// TIA Portal V19 export
FUNCTION "FC40_CommSlave" : Void   // FC40, LAD
{ S7_Optimized_Access := 'TRUE' }
// stored: AutoNumber false, IsIECCheckEnabled true, SetENOAutomatically false
BEGIN

REGION Network 1: Manage communication with Left PLC
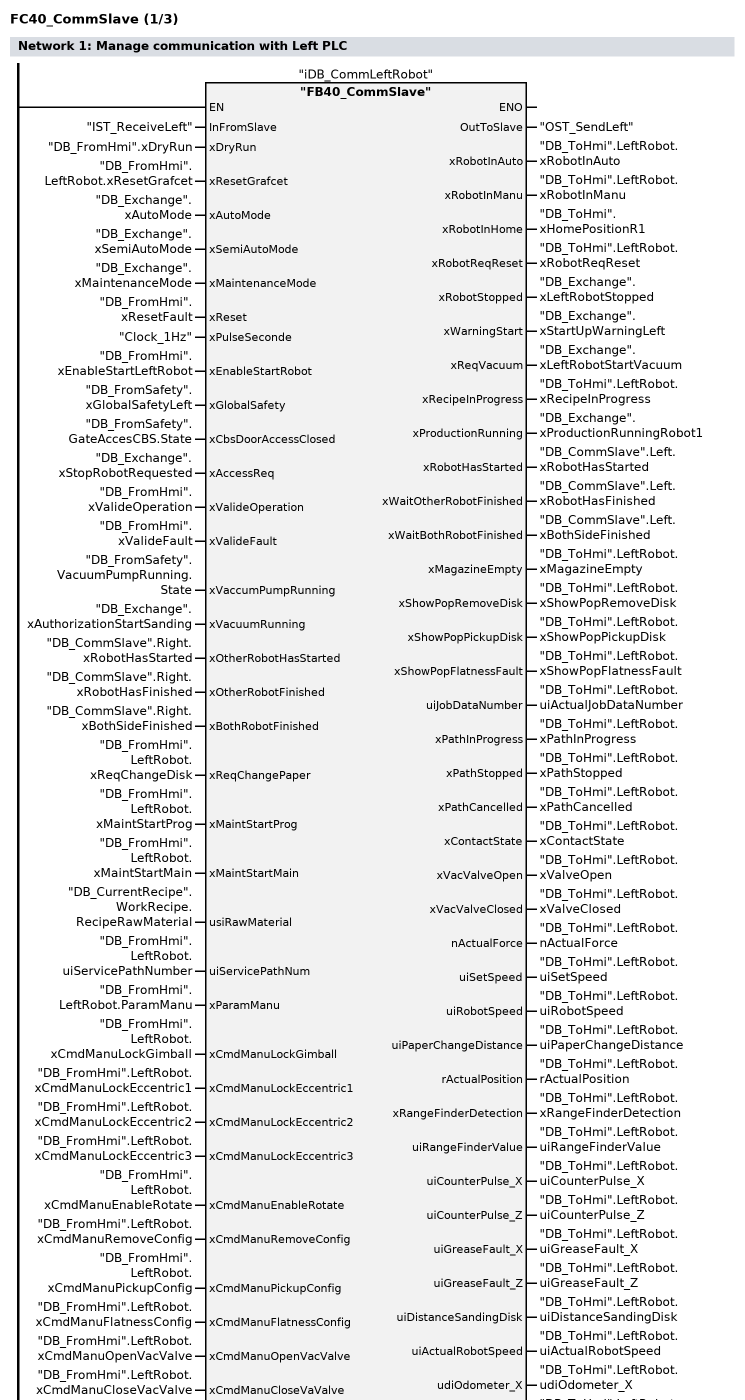
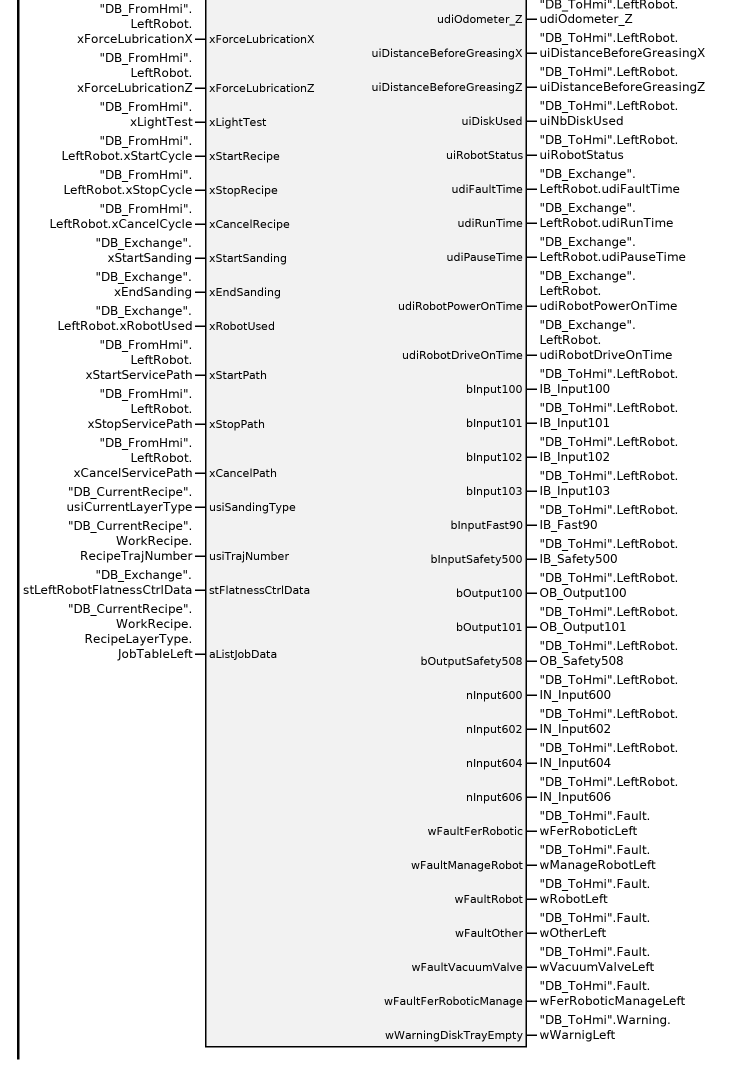
   RUNG wire#powerrail
      "iDB_CommLeftRobot"(InFromSlave := "IST_ReceiveLeft", xDryRun := "DB_FromHmi".xDryRun, xResetGrafcet := "DB_FromHmi".LeftRobot.xResetGrafcet, xAutoMode := "DB_Exchange".xAutoMode, xSemiAutoMode := "DB_Exchange".xSemiAutoMode, xMaintenanceMode := "DB_Exchange".xMaintenanceMode, xReset := "DB_FromHmi".xResetFault, xPulseSeconde := "Clock_1Hz", xEnableStartRobot := "DB_FromHmi".xEnableStartLeftRobot, xGlobalSafety := "DB_FromSafety".xGlobalSafetyLeft, xCbsDoorAccessClosed := "DB_FromSafety".GateAccesCBS.State, xAccessReq := "DB_Exchange".xStopRobotRequested, xValideOperation := "DB_FromHmi".xValideOperation, xValideFault := "DB_FromHmi".xValideFault, xVaccumPumpRunning := "DB_FromSafety".VacuumPumpRunning.State, xVacuumRunning := "DB_Exchange".xAuthorizationStartSanding, xOtherRobotHasStarted := "DB_CommSlave".Right.xRobotHasStarted, xOtherRobotFinished := "DB_CommSlave".Right.xRobotHasFinished, xBothRobotFinished := "DB_CommSlave".Right.xBothSideFinished, xReqChangePaper := "DB_FromHmi".LeftRobot.xReqChangeDisk, xMaintStartProg := "DB_FromHmi".LeftRobot.xMaintStartProg, xMaintStartMain := "DB_FromHmi".LeftRobot.xMaintStartMain, usiRawMaterial := "DB_CurrentRecipe".WorkRecipe.RecipeRawMaterial, uiServicePathNum := "DB_FromHmi".LeftRobot.uiServicePathNumber, xParamManu := "DB_FromHmi".LeftRobot.ParamManu, xCmdManuLockGimball := "DB_FromHmi".LeftRobot.xCmdManuLockGimball, xCmdManuLockEccentric1 := "DB_FromHmi".LeftRobot.xCmdManuLockEccentric1, xCmdManuLockEccentric2 := "DB_FromHmi".LeftRobot.xCmdManuLockEccentric2, xCmdManuLockEccentric3 := "DB_FromHmi".LeftRobot.xCmdManuLockEccentric3, xCmdManuEnableRotate := "DB_FromHmi".LeftRobot.xCmdManuEnableRotate, xCmdManuRemoveConfig := "DB_FromHmi".LeftRobot.xCmdManuRemoveConfig, xCmdManuPickupConfig := "DB_FromHmi".LeftRobot.xCmdManuPickupConfig, xCmdManuFlatnessConfig := "DB_FromHmi".LeftRobot.xCmdManuFlatnessConfig, xCmdManuOpenVacValve := "DB_FromHmi".LeftRobot.xCmdManuOpenVacValve, xCmdManuCloseVaValve := "DB_FromHmi".LeftRobot.xCmdManuCloseVacValve, xForceLubricationX := "DB_FromHmi".LeftRobot.xForceLubricationX, xForceLubricationZ := "DB_FromHmi".LeftRobot.xForceLubricationZ, xLightTest := "DB_FromHmi".xLightTest, xStartRecipe := "DB_FromHmi".LeftRobot.xStartCycle, xStopRecipe := "DB_FromHmi".LeftRobot.xStopCycle, xCancelRecipe := "DB_FromHmi".LeftRobot.xCancelCycle, xStartSanding := "DB_Exchange".xStartSanding, xEndSanding := "DB_Exchange".xEndSanding, xRobotUsed := "DB_Exchange".LeftRobot.xRobotUsed, xStartPath := "DB_FromHmi".LeftRobot.xStartServicePath, xStopPath := "DB_FromHmi".LeftRobot.xStopServicePath, xCancelPath := "DB_FromHmi".LeftRobot.xCancelServicePath, usiSandingType := "DB_CurrentRecipe".usiCurrentLayerType, usiTrajNumber := "DB_CurrentRecipe".WorkRecipe.RecipeTrajNumber, stFlatnessCtrlData := "DB_Exchange".stLeftRobotFlatnessCtrlData, aListJobData := "DB_CurrentRecipe".WorkRecipe.RecipeLayerType.JobTableLeft, OutToSlave => "OST_SendLeft", xRobotInAuto => "DB_ToHmi".LeftRobot.xRobotInAuto, xRobotInManu => "DB_ToHmi".LeftRobot.xRobotInManu, xRobotInHome => "DB_ToHmi".xHomePositionR1, xRobotReqReset => "DB_ToHmi".LeftRobot.xRobotReqReset, xRobotStopped => "DB_Exchange".xLeftRobotStopped, xWarningStart => "DB_Exchange".xStartUpWarningLeft, xReqVacuum => "DB_Exchange".xLeftRobotStartVacuum, xRecipeInProgress => "DB_ToHmi".LeftRobot.xRecipeInProgress, xProductionRunning => "DB_Exchange".xProductionRunningRobot1, xRobotHasStarted => "DB_CommSlave".Left.xRobotHasStarted, xWaitOtherRobotFinished => "DB_CommSlave".Left.xRobotHasFinished, xWaitBothRobotFinished => "DB_CommSlave".Left.xBothSideFinished, xMagazineEmpty => "DB_ToHmi".LeftRobot.xMagazineEmpty, xShowPopRemoveDisk => "DB_ToHmi".LeftRobot.xShowPopRemoveDisk, xShowPopPickupDisk => "DB_ToHmi".LeftRobot.xShowPopPickupDisk, xShowPopFlatnessFault => "DB_ToHmi".LeftRobot.xShowPopFlatnessFault, uiJobDataNumber => "DB_ToHmi".LeftRobot.uiActualJobDataNumber, xPathInProgress => "DB_ToHmi".LeftRobot.xPathInProgress, xPathStopped => "DB_ToHmi".LeftRobot.xPathStopped, xPathCancelled => "DB_ToHmi".LeftRobot.xPathCancelled, xContactState => "DB_ToHmi".LeftRobot.xContactState, xVacValveOpen => "DB_ToHmi".LeftRobot.xValveOpen, xVacValveClosed => "DB_ToHmi".LeftRobot.xValveClosed, nActualForce => "DB_ToHmi".LeftRobot.nActualForce, uiSetSpeed => "DB_ToHmi".LeftRobot.uiSetSpeed, uiRobotSpeed => "DB_ToHmi".LeftRobot.uiRobotSpeed, uiPaperChangeDistance => "DB_ToHmi".LeftRobot.uiPaperChangeDistance, rActualPosition => "DB_ToHmi".LeftRobot.rActualPosition, xRangeFinderDetection => "DB_ToHmi".LeftRobot.xRangeFinderDetection, uiRangeFinderValue => "DB_ToHmi".LeftRobot.uiRangeFinderValue, uiCounterPulse_X => "DB_ToHmi".LeftRobot.uiCounterPulse_X, uiCounterPulse_Z => "DB_ToHmi".LeftRobot.uiCounterPulse_Z, uiGreaseFault_X => "DB_ToHmi".LeftRobot.uiGreaseFault_X, uiGreaseFault_Z => "DB_ToHmi".LeftRobot.uiGreaseFault_Z, uiDistanceSandingDisk => "DB_ToHmi".LeftRobot.uiDistanceSandingDisk, uiActualRobotSpeed => "DB_ToHmi".LeftRobot.uiActualRobotSpeed, udiOdometer_X => "DB_ToHmi".LeftRobot.udiOdometer_X, udiOdometer_Z => "DB_ToHmi".LeftRobot.udiOdometer_Z, uiDistanceBeforeGreasingX => "DB_ToHmi".LeftRobot.uiDistanceBeforeGreasingX, uiDistanceBeforeGreasingZ => "DB_ToHmi".LeftRobot.uiDistanceBeforeGreasingZ, uiDiskUsed => "DB_ToHmi".LeftRobot.uiNbDiskUsed, uiRobotStatus => "DB_ToHmi".LeftRobot.uiRobotStatus, udiFaultTime => "DB_Exchange".LeftRobot.udiFaultTime, udiRunTime => "DB_Exchange".LeftRobot.udiRunTime, udiPauseTime => "DB_Exchange".LeftRobot.udiPauseTime, udiRobotPowerOnTime => "DB_Exchange".LeftRobot.udiRobotPowerOnTime, udiRobotDriveOnTime => "DB_Exchange".LeftRobot.udiRobotDriveOnTime, bInput100 => "DB_ToHmi".LeftRobot.IB_Input100, bInput101 => "DB_ToHmi".LeftRobot.IB_Input101, bInput102 => "DB_ToHmi".LeftRobot.IB_Input102, bInput103 => "DB_ToHmi".LeftRobot.IB_Input103, bInputFast90 => "DB_ToHmi".LeftRobot.IB_Fast90, bInputSafety500 => "DB_ToHmi".LeftRobot.IB_Safety500, bOutput100 => "DB_ToHmi".LeftRobot.OB_Output100, bOutput101 => "DB_ToHmi".LeftRobot.OB_Output101, bOutputSafety508 => "DB_ToHmi".LeftRobot.OB_Safety508, nInput600 => "DB_ToHmi".LeftRobot.IN_Input600, nInput602 => "DB_ToHmi".LeftRobot.IN_Input602, nInput604 => "DB_ToHmi".LeftRobot.IN_Input604, nInput606 => "DB_ToHmi".LeftRobot.IN_Input606, wFaultFerRobotic => "DB_ToHmi".Fault.wFerRoboticLeft, wFaultManageRobot => "DB_ToHmi".Fault.wManageRobotLeft, wFaultRobot => "DB_ToHmi".Fault.wRobotLeft, wFaultOther => "DB_ToHmi".Fault.wOtherLeft, wFaultVacuumValve => "DB_ToHmi".Fault.wVacuumValveLeft, wFaultFerRoboticManage => "DB_ToHmi".Fault.wFerRoboticManageLeft, wWarningDiskTrayEmpty => "DB_ToHmi".Warning.wWarnigLeft)
   END_RUNG
   // the same network as SCL:
   "iDB_CommLeftRobot"(InFromSlave := "IST_ReceiveLeft",   // "FB40_CommSlave"
                       xDryRun := "DB_FromHmi".xDryRun,
                       xResetGrafcet := "DB_FromHmi".LeftRobot.xResetGrafcet,
                       xAutoMode := "DB_Exchange".xAutoMode,
                       xSemiAutoMode := "DB_Exchange".xSemiAutoMode,
                       xMaintenanceMode := "DB_Exchange".xMaintenanceMode,
                       xReset := "DB_FromHmi".xResetFault,
                       xPulseSeconde := "Clock_1Hz",
                       xEnableStartRobot := "DB_FromHmi".xEnableStartLeftRobot,
                       xGlobalSafety := "DB_FromSafety".xGlobalSafetyLeft,
                       xCbsDoorAccessClosed := "DB_FromSafety".GateAccesCBS.State,
                       xAccessReq := "DB_Exchange".xStopRobotRequested,
                       xValideOperation := "DB_FromHmi".xValideOperation,
                       xValideFault := "DB_FromHmi".xValideFault,
                       xVaccumPumpRunning := "DB_FromSafety".VacuumPumpRunning.State,
                       xVacuumRunning := "DB_Exchange".xAuthorizationStartSanding,
                       xOtherRobotHasStarted := "DB_CommSlave".Right.xRobotHasStarted,
                       xOtherRobotFinished := "DB_CommSlave".Right.xRobotHasFinished,
                       xBothRobotFinished := "DB_CommSlave".Right.xBothSideFinished,
                       xReqChangePaper := "DB_FromHmi".LeftRobot.xReqChangeDisk,
                       xMaintStartProg := "DB_FromHmi".LeftRobot.xMaintStartProg,
                       xMaintStartMain := "DB_FromHmi".LeftRobot.xMaintStartMain,
                       usiRawMaterial := "DB_CurrentRecipe".WorkRecipe.RecipeRawMaterial,
                       uiServicePathNum := "DB_FromHmi".LeftRobot.uiServicePathNumber,
                       xParamManu := "DB_FromHmi".LeftRobot.ParamManu,
                       xCmdManuLockGimball := "DB_FromHmi".LeftRobot.xCmdManuLockGimball,
                       xCmdManuLockEccentric1 := "DB_FromHmi".LeftRobot.xCmdManuLockEccentric1,
                       xCmdManuLockEccentric2 := "DB_FromHmi".LeftRobot.xCmdManuLockEccentric2,
                       xCmdManuLockEccentric3 := "DB_FromHmi".LeftRobot.xCmdManuLockEccentric3,
                       xCmdManuEnableRotate := "DB_FromHmi".LeftRobot.xCmdManuEnableRotate,
                       xCmdManuRemoveConfig := "DB_FromHmi".LeftRobot.xCmdManuRemoveConfig,
                       xCmdManuPickupConfig := "DB_FromHmi".LeftRobot.xCmdManuPickupConfig,
                       xCmdManuFlatnessConfig := "DB_FromHmi".LeftRobot.xCmdManuFlatnessConfig,
                       xCmdManuOpenVacValve := "DB_FromHmi".LeftRobot.xCmdManuOpenVacValve,
                       xCmdManuCloseVaValve := "DB_FromHmi".LeftRobot.xCmdManuCloseVacValve,
                       xForceLubricationX := "DB_FromHmi".LeftRobot.xForceLubricationX,
                       xForceLubricationZ := "DB_FromHmi".LeftRobot.xForceLubricationZ,
                       xLightTest := "DB_FromHmi".xLightTest,
                       xStartRecipe := "DB_FromHmi".LeftRobot.xStartCycle,
                       xStopRecipe := "DB_FromHmi".LeftRobot.xStopCycle,
                       xCancelRecipe := "DB_FromHmi".LeftRobot.xCancelCycle,
                       xStartSanding := "DB_Exchange".xStartSanding,
                       xEndSanding := "DB_Exchange".xEndSanding,
                       xRobotUsed := "DB_Exchange".LeftRobot.xRobotUsed,
                       xStartPath := "DB_FromHmi".LeftRobot.xStartServicePath,
                       xStopPath := "DB_FromHmi".LeftRobot.xStopServicePath,
                       xCancelPath := "DB_FromHmi".LeftRobot.xCancelServicePath,
                       usiSandingType := "DB_CurrentRecipe".usiCurrentLayerType,
                       usiTrajNumber := "DB_CurrentRecipe".WorkRecipe.RecipeTrajNumber,
                       stFlatnessCtrlData := "DB_Exchange".stLeftRobotFlatnessCtrlData,
                       aListJobData := "DB_CurrentRecipe".WorkRecipe.RecipeLayerType.JobTableLeft,
                       OutToSlave => "OST_SendLeft",
                       xRobotInAuto => "DB_ToHmi".LeftRobot.xRobotInAuto,
                       xRobotInManu => "DB_ToHmi".LeftRobot.xRobotInManu,
                       xRobotInHome => "DB_ToHmi".xHomePositionR1,
                       xRobotReqReset => "DB_ToHmi".LeftRobot.xRobotReqReset,
                       xRobotStopped => "DB_Exchange".xLeftRobotStopped,
                       xWarningStart => "DB_Exchange".xStartUpWarningLeft,
                       xReqVacuum => "DB_Exchange".xLeftRobotStartVacuum,
                       xRecipeInProgress => "DB_ToHmi".LeftRobot.xRecipeInProgress,
                       xProductionRunning => "DB_Exchange".xProductionRunningRobot1,
                       xRobotHasStarted => "DB_CommSlave".Left.xRobotHasStarted,
                       xWaitOtherRobotFinished => "DB_CommSlave".Left.xRobotHasFinished,
                       xWaitBothRobotFinished => "DB_CommSlave".Left.xBothSideFinished,
                       xMagazineEmpty => "DB_ToHmi".LeftRobot.xMagazineEmpty,
                       xShowPopRemoveDisk => "DB_ToHmi".LeftRobot.xShowPopRemoveDisk,
                       xShowPopPickupDisk => "DB_ToHmi".LeftRobot.xShowPopPickupDisk,
                       xShowPopFlatnessFault => "DB_ToHmi".LeftRobot.xShowPopFlatnessFault,
                       uiJobDataNumber => "DB_ToHmi".LeftRobot.uiActualJobDataNumber,
                       xPathInProgress => "DB_ToHmi".LeftRobot.xPathInProgress,
                       xPathStopped => "DB_ToHmi".LeftRobot.xPathStopped,
                       xPathCancelled => "DB_ToHmi".LeftRobot.xPathCancelled,
                       xContactState => "DB_ToHmi".LeftRobot.xContactState,
                       xVacValveOpen => "DB_ToHmi".LeftRobot.xValveOpen,
                       xVacValveClosed => "DB_ToHmi".LeftRobot.xValveClosed,
                       nActualForce => "DB_ToHmi".LeftRobot.nActualForce,
                       uiSetSpeed => "DB_ToHmi".LeftRobot.uiSetSpeed,
                       uiRobotSpeed => "DB_ToHmi".LeftRobot.uiRobotSpeed,
                       uiPaperChangeDistance => "DB_ToHmi".LeftRobot.uiPaperChangeDistance,
                       rActualPosition => "DB_ToHmi".LeftRobot.rActualPosition,
                       xRangeFinderDetection => "DB_ToHmi".LeftRobot.xRangeFinderDetection,
                       uiRangeFinderValue => "DB_ToHmi".LeftRobot.uiRangeFinderValue,
                       uiCounterPulse_X => "DB_ToHmi".LeftRobot.uiCounterPulse_X,
                       uiCounterPulse_Z => "DB_ToHmi".LeftRobot.uiCounterPulse_Z,
                       uiGreaseFault_X => "DB_ToHmi".LeftRobot.uiGreaseFault_X,
                       uiGreaseFault_Z => "DB_ToHmi".LeftRobot.uiGreaseFault_Z,
                       uiDistanceSandingDisk => "DB_ToHmi".LeftRobot.uiDistanceSandingDisk,
                       uiActualRobotSpeed => "DB_ToHmi".LeftRobot.uiActualRobotSpeed,
                       udiOdometer_X => "DB_ToHmi".LeftRobot.udiOdometer_X,
                       udiOdometer_Z => "DB_ToHmi".LeftRobot.udiOdometer_Z,
                       uiDistanceBeforeGreasingX => "DB_ToHmi".LeftRobot.uiDistanceBeforeGreasingX,
                       uiDistanceBeforeGreasingZ => "DB_ToHmi".LeftRobot.uiDistanceBeforeGreasingZ,
                       uiDiskUsed => "DB_ToHmi".LeftRobot.uiNbDiskUsed,
                       uiRobotStatus => "DB_ToHmi".LeftRobot.uiRobotStatus,
                       udiFaultTime => "DB_Exchange".LeftRobot.udiFaultTime,
                       udiRunTime => "DB_Exchange".LeftRobot.udiRunTime,
                       udiPauseTime => "DB_Exchange".LeftRobot.udiPauseTime,
                       udiRobotPowerOnTime => "DB_Exchange".LeftRobot.udiRobotPowerOnTime,
                       udiRobotDriveOnTime => "DB_Exchange".LeftRobot.udiRobotDriveOnTime,
                       bInput100 => "DB_ToHmi".LeftRobot.IB_Input100,
                       bInput101 => "DB_ToHmi".LeftRobot.IB_Input101,
                       bInput102 => "DB_ToHmi".LeftRobot.IB_Input102,
                       bInput103 => "DB_ToHmi".LeftRobot.IB_Input103,
                       bInputFast90 => "DB_ToHmi".LeftRobot.IB_Fast90,
                       bInputSafety500 => "DB_ToHmi".LeftRobot.IB_Safety500,
                       bOutput100 => "DB_ToHmi".LeftRobot.OB_Output100,
                       bOutput101 => "DB_ToHmi".LeftRobot.OB_Output101,
                       bOutputSafety508 => "DB_ToHmi".LeftRobot.OB_Safety508,
                       nInput600 => "DB_ToHmi".LeftRobot.IN_Input600,
                       nInput602 => "DB_ToHmi".LeftRobot.IN_Input602,
                       nInput604 => "DB_ToHmi".LeftRobot.IN_Input604,
                       nInput606 => "DB_ToHmi".LeftRobot.IN_Input606,
                       wFaultFerRobotic => "DB_ToHmi".Fault.wFerRoboticLeft,
                       wFaultManageRobot => "DB_ToHmi".Fault.wManageRobotLeft,
                       wFaultRobot => "DB_ToHmi".Fault.wRobotLeft,
                       wFaultOther => "DB_ToHmi".Fault.wOtherLeft,
                       wFaultVacuumValve => "DB_ToHmi".Fault.wVacuumValveLeft,
                       wFaultFerRoboticManage => "DB_ToHmi".Fault.wFerRoboticManageLeft,
                       wWarningDiskTrayEmpty => "DB_ToHmi".Warning.wWarnigLeft);
END_REGION

REGION Network 2: Manage communication with Right PLC
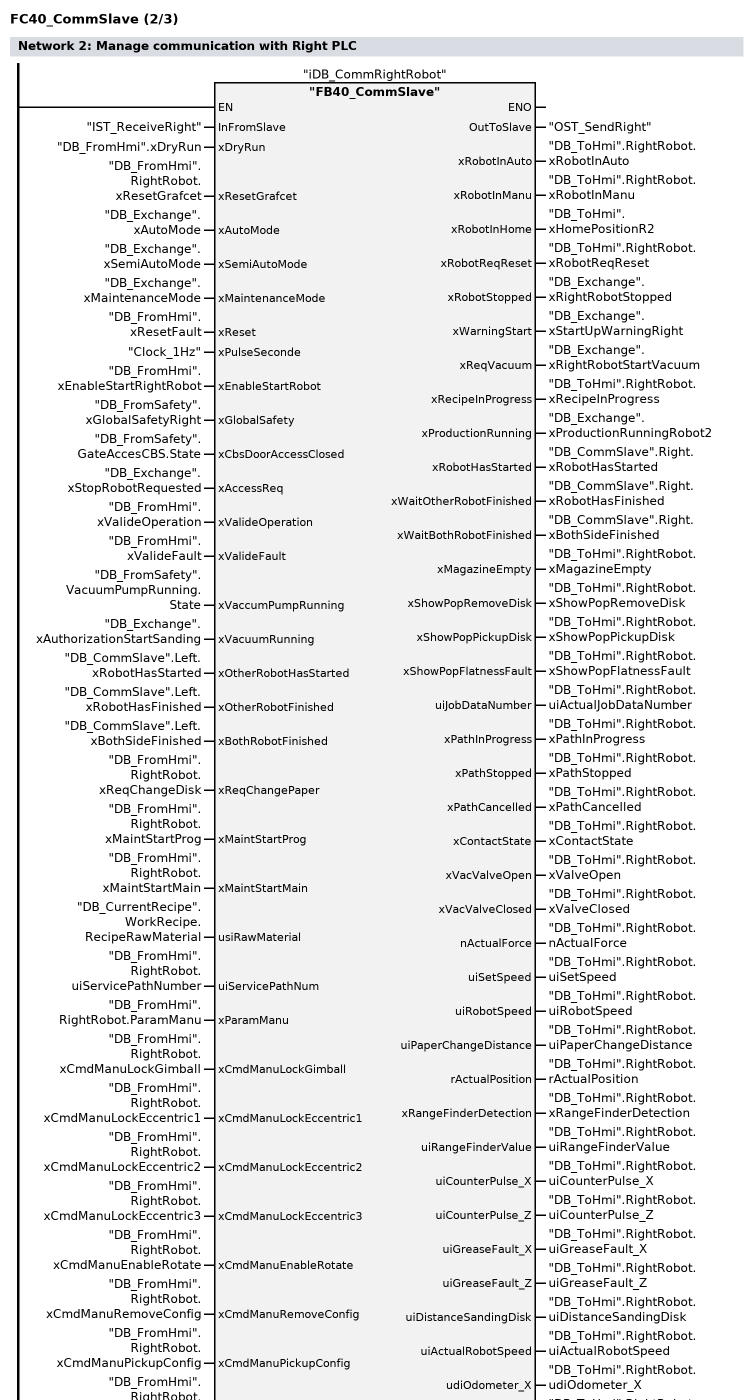
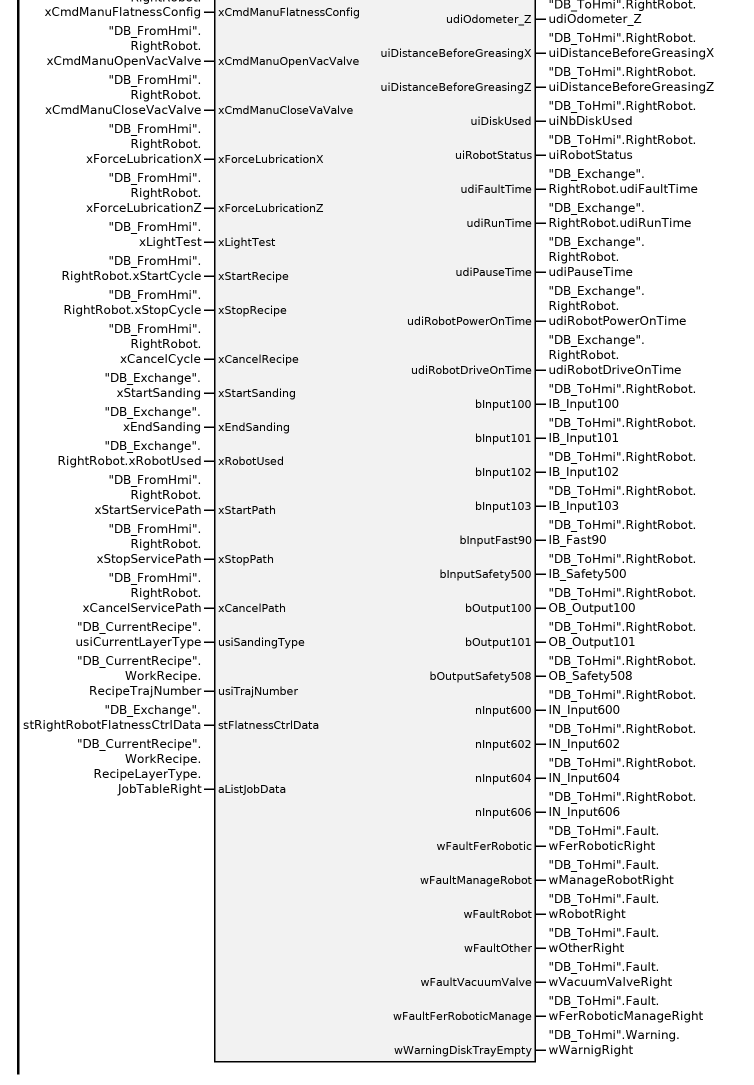
   RUNG wire#powerrail
      "iDB_CommRightRobot"(InFromSlave := "IST_ReceiveRight", xDryRun := "DB_FromHmi".xDryRun, xResetGrafcet := "DB_FromHmi".RightRobot.xResetGrafcet, xAutoMode := "DB_Exchange".xAutoMode, xSemiAutoMode := "DB_Exchange".xSemiAutoMode, xMaintenanceMode := "DB_Exchange".xMaintenanceMode, xReset := "DB_FromHmi".xResetFault, xPulseSeconde := "Clock_1Hz", xEnableStartRobot := "DB_FromHmi".xEnableStartRightRobot, xGlobalSafety := "DB_FromSafety".xGlobalSafetyRight, xCbsDoorAccessClosed := "DB_FromSafety".GateAccesCBS.State, xAccessReq := "DB_Exchange".xStopRobotRequested, xValideOperation := "DB_FromHmi".xValideOperation, xValideFault := "DB_FromHmi".xValideFault, xVaccumPumpRunning := "DB_FromSafety".VacuumPumpRunning.State, xVacuumRunning := "DB_Exchange".xAuthorizationStartSanding, xOtherRobotHasStarted := "DB_CommSlave".Left.xRobotHasStarted, xOtherRobotFinished := "DB_CommSlave".Left.xRobotHasFinished, xBothRobotFinished := "DB_CommSlave".Left.xBothSideFinished, xReqChangePaper := "DB_FromHmi".RightRobot.xReqChangeDisk, xMaintStartProg := "DB_FromHmi".RightRobot.xMaintStartProg, xMaintStartMain := "DB_FromHmi".RightRobot.xMaintStartMain, usiRawMaterial := "DB_CurrentRecipe".WorkRecipe.RecipeRawMaterial, uiServicePathNum := "DB_FromHmi".RightRobot.uiServicePathNumber, xParamManu := "DB_FromHmi".RightRobot.ParamManu, xCmdManuLockGimball := "DB_FromHmi".RightRobot.xCmdManuLockGimball, xCmdManuLockEccentric1 := "DB_FromHmi".RightRobot.xCmdManuLockEccentric1, xCmdManuLockEccentric2 := "DB_FromHmi".RightRobot.xCmdManuLockEccentric2, xCmdManuLockEccentric3 := "DB_FromHmi".RightRobot.xCmdManuLockEccentric3, xCmdManuEnableRotate := "DB_FromHmi".RightRobot.xCmdManuEnableRotate, xCmdManuRemoveConfig := "DB_FromHmi".RightRobot.xCmdManuRemoveConfig, xCmdManuPickupConfig := "DB_FromHmi".RightRobot.xCmdManuPickupConfig, xCmdManuFlatnessConfig := "DB_FromHmi".RightRobot.xCmdManuFlatnessConfig, xCmdManuOpenVacValve := "DB_FromHmi".RightRobot.xCmdManuOpenVacValve, xCmdManuCloseVaValve := "DB_FromHmi".RightRobot.xCmdManuCloseVacValve, xForceLubricationX := "DB_FromHmi".RightRobot.xForceLubricationX, xForceLubricationZ := "DB_FromHmi".RightRobot.xForceLubricationZ, xLightTest := "DB_FromHmi".xLightTest, xStartRecipe := "DB_FromHmi".RightRobot.xStartCycle, xStopRecipe := "DB_FromHmi".RightRobot.xStopCycle, xCancelRecipe := "DB_FromHmi".RightRobot.xCancelCycle, xStartSanding := "DB_Exchange".xStartSanding, xEndSanding := "DB_Exchange".xEndSanding, xRobotUsed := "DB_Exchange".RightRobot.xRobotUsed, xStartPath := "DB_FromHmi".RightRobot.xStartServicePath, xStopPath := "DB_FromHmi".RightRobot.xStopServicePath, xCancelPath := "DB_FromHmi".RightRobot.xCancelServicePath, usiSandingType := "DB_CurrentRecipe".usiCurrentLayerType, usiTrajNumber := "DB_CurrentRecipe".WorkRecipe.RecipeTrajNumber, stFlatnessCtrlData := "DB_Exchange".stRightRobotFlatnessCtrlData, aListJobData := "DB_CurrentRecipe".WorkRecipe.RecipeLayerType.JobTableRight, OutToSlave => "OST_SendRight", xRobotInAuto => "DB_ToHmi".RightRobot.xRobotInAuto, xRobotInManu => "DB_ToHmi".RightRobot.xRobotInManu, xRobotInHome => "DB_ToHmi".xHomePositionR2, xRobotReqReset => "DB_ToHmi".RightRobot.xRobotReqReset, xRobotStopped => "DB_Exchange".xRightRobotStopped, xWarningStart => "DB_Exchange".xStartUpWarningRight, xReqVacuum => "DB_Exchange".xRightRobotStartVacuum, xRecipeInProgress => "DB_ToHmi".RightRobot.xRecipeInProgress, xProductionRunning => "DB_Exchange".xProductionRunningRobot2, xRobotHasStarted => "DB_CommSlave".Right.xRobotHasStarted, xWaitOtherRobotFinished => "DB_CommSlave".Right.xRobotHasFinished, xWaitBothRobotFinished => "DB_CommSlave".Right.xBothSideFinished, xMagazineEmpty => "DB_ToHmi".RightRobot.xMagazineEmpty, xShowPopRemoveDisk => "DB_ToHmi".RightRobot.xShowPopRemoveDisk, xShowPopPickupDisk => "DB_ToHmi".RightRobot.xShowPopPickupDisk, xShowPopFlatnessFault => "DB_ToHmi".RightRobot.xShowPopFlatnessFault, uiJobDataNumber => "DB_ToHmi".RightRobot.uiActualJobDataNumber, xPathInProgress => "DB_ToHmi".RightRobot.xPathInProgress, xPathStopped => "DB_ToHmi".RightRobot.xPathStopped, xPathCancelled => "DB_ToHmi".RightRobot.xPathCancelled, xContactState => "DB_ToHmi".RightRobot.xContactState, xVacValveOpen => "DB_ToHmi".RightRobot.xValveOpen, xVacValveClosed => "DB_ToHmi".RightRobot.xValveClosed, nActualForce => "DB_ToHmi".RightRobot.nActualForce, uiSetSpeed => "DB_ToHmi".RightRobot.uiSetSpeed, uiRobotSpeed => "DB_ToHmi".RightRobot.uiRobotSpeed, uiPaperChangeDistance => "DB_ToHmi".RightRobot.uiPaperChangeDistance, rActualPosition => "DB_ToHmi".RightRobot.rActualPosition, xRangeFinderDetection => "DB_ToHmi".RightRobot.xRangeFinderDetection, uiRangeFinderValue => "DB_ToHmi".RightRobot.uiRangeFinderValue, uiCounterPulse_X => "DB_ToHmi".RightRobot.uiCounterPulse_X, uiCounterPulse_Z => "DB_ToHmi".RightRobot.uiCounterPulse_Z, uiGreaseFault_X => "DB_ToHmi".RightRobot.uiGreaseFault_X, uiGreaseFault_Z => "DB_ToHmi".RightRobot.uiGreaseFault_Z, uiDistanceSandingDisk => "DB_ToHmi".RightRobot.uiDistanceSandingDisk, uiActualRobotSpeed => "DB_ToHmi".RightRobot.uiActualRobotSpeed, udiOdometer_X => "DB_ToHmi".RightRobot.udiOdometer_X, udiOdometer_Z => "DB_ToHmi".RightRobot.udiOdometer_Z, uiDistanceBeforeGreasingX => "DB_ToHmi".RightRobot.uiDistanceBeforeGreasingX, uiDistanceBeforeGreasingZ => "DB_ToHmi".RightRobot.uiDistanceBeforeGreasingZ, uiDiskUsed => "DB_ToHmi".RightRobot.uiNbDiskUsed, uiRobotStatus => "DB_ToHmi".RightRobot.uiRobotStatus, udiFaultTime => "DB_Exchange".RightRobot.udiFaultTime, udiRunTime => "DB_Exchange".RightRobot.udiRunTime, udiPauseTime => "DB_Exchange".RightRobot.udiPauseTime, udiRobotPowerOnTime => "DB_Exchange".RightRobot.udiRobotPowerOnTime, udiRobotDriveOnTime => "DB_Exchange".RightRobot.udiRobotDriveOnTime, bInput100 => "DB_ToHmi".RightRobot.IB_Input100, bInput101 => "DB_ToHmi".RightRobot.IB_Input101, bInput102 => "DB_ToHmi".RightRobot.IB_Input102, bInput103 => "DB_ToHmi".RightRobot.IB_Input103, bInputFast90 => "DB_ToHmi".RightRobot.IB_Fast90, bInputSafety500 => "DB_ToHmi".RightRobot.IB_Safety500, bOutput100 => "DB_ToHmi".RightRobot.OB_Output100, bOutput101 => "DB_ToHmi".RightRobot.OB_Output101, bOutputSafety508 => "DB_ToHmi".RightRobot.OB_Safety508, nInput600 => "DB_ToHmi".RightRobot.IN_Input600, nInput602 => "DB_ToHmi".RightRobot.IN_Input602, nInput604 => "DB_ToHmi".RightRobot.IN_Input604, nInput606 => "DB_ToHmi".RightRobot.IN_Input606, wFaultFerRobotic => "DB_ToHmi".Fault.wFerRoboticRight, wFaultManageRobot => "DB_ToHmi".Fault.wManageRobotRight, wFaultRobot => "DB_ToHmi".Fault.wRobotRight, wFaultOther => "DB_ToHmi".Fault.wOtherRight, wFaultVacuumValve => "DB_ToHmi".Fault.wVacuumValveRight, wFaultFerRoboticManage => "DB_ToHmi".Fault.wFerRoboticManageRight, wWarningDiskTrayEmpty => "DB_ToHmi".Warning.wWarnigRight)
   END_RUNG
   // the same network as SCL:
   "iDB_CommRightRobot"(InFromSlave := "IST_ReceiveRight",   // "FB40_CommSlave"
                        xDryRun := "DB_FromHmi".xDryRun,
                        xResetGrafcet := "DB_FromHmi".RightRobot.xResetGrafcet,
                        xAutoMode := "DB_Exchange".xAutoMode,
                        xSemiAutoMode := "DB_Exchange".xSemiAutoMode,
                        xMaintenanceMode := "DB_Exchange".xMaintenanceMode,
                        xReset := "DB_FromHmi".xResetFault,
                        xPulseSeconde := "Clock_1Hz",
                        xEnableStartRobot := "DB_FromHmi".xEnableStartRightRobot,
                        xGlobalSafety := "DB_FromSafety".xGlobalSafetyRight,
                        xCbsDoorAccessClosed := "DB_FromSafety".GateAccesCBS.State,
                        xAccessReq := "DB_Exchange".xStopRobotRequested,
                        xValideOperation := "DB_FromHmi".xValideOperation,
                        xValideFault := "DB_FromHmi".xValideFault,
                        xVaccumPumpRunning := "DB_FromSafety".VacuumPumpRunning.State,
                        xVacuumRunning := "DB_Exchange".xAuthorizationStartSanding,
                        xOtherRobotHasStarted := "DB_CommSlave".Left.xRobotHasStarted,
                        xOtherRobotFinished := "DB_CommSlave".Left.xRobotHasFinished,
                        xBothRobotFinished := "DB_CommSlave".Left.xBothSideFinished,
                        xReqChangePaper := "DB_FromHmi".RightRobot.xReqChangeDisk,
                        xMaintStartProg := "DB_FromHmi".RightRobot.xMaintStartProg,
                        xMaintStartMain := "DB_FromHmi".RightRobot.xMaintStartMain,
                        usiRawMaterial := "DB_CurrentRecipe".WorkRecipe.RecipeRawMaterial,
                        uiServicePathNum := "DB_FromHmi".RightRobot.uiServicePathNumber,
                        xParamManu := "DB_FromHmi".RightRobot.ParamManu,
                        xCmdManuLockGimball := "DB_FromHmi".RightRobot.xCmdManuLockGimball,
                        xCmdManuLockEccentric1 := "DB_FromHmi".RightRobot.xCmdManuLockEccentric1,
                        xCmdManuLockEccentric2 := "DB_FromHmi".RightRobot.xCmdManuLockEccentric2,
                        xCmdManuLockEccentric3 := "DB_FromHmi".RightRobot.xCmdManuLockEccentric3,
                        xCmdManuEnableRotate := "DB_FromHmi".RightRobot.xCmdManuEnableRotate,
                        xCmdManuRemoveConfig := "DB_FromHmi".RightRobot.xCmdManuRemoveConfig,
                        xCmdManuPickupConfig := "DB_FromHmi".RightRobot.xCmdManuPickupConfig,
                        xCmdManuFlatnessConfig := "DB_FromHmi".RightRobot.xCmdManuFlatnessConfig,
                        xCmdManuOpenVacValve := "DB_FromHmi".RightRobot.xCmdManuOpenVacValve,
                        xCmdManuCloseVaValve := "DB_FromHmi".RightRobot.xCmdManuCloseVacValve,
                        xForceLubricationX := "DB_FromHmi".RightRobot.xForceLubricationX,
                        xForceLubricationZ := "DB_FromHmi".RightRobot.xForceLubricationZ,
                        xLightTest := "DB_FromHmi".xLightTest,
                        xStartRecipe := "DB_FromHmi".RightRobot.xStartCycle,
                        xStopRecipe := "DB_FromHmi".RightRobot.xStopCycle,
                        xCancelRecipe := "DB_FromHmi".RightRobot.xCancelCycle,
                        xStartSanding := "DB_Exchange".xStartSanding,
                        xEndSanding := "DB_Exchange".xEndSanding,
                        xRobotUsed := "DB_Exchange".RightRobot.xRobotUsed,
                        xStartPath := "DB_FromHmi".RightRobot.xStartServicePath,
                        xStopPath := "DB_FromHmi".RightRobot.xStopServicePath,
                        xCancelPath := "DB_FromHmi".RightRobot.xCancelServicePath,
                        usiSandingType := "DB_CurrentRecipe".usiCurrentLayerType,
                        usiTrajNumber := "DB_CurrentRecipe".WorkRecipe.RecipeTrajNumber,
                        stFlatnessCtrlData := "DB_Exchange".stRightRobotFlatnessCtrlData,
                        aListJobData := "DB_CurrentRecipe".WorkRecipe.RecipeLayerType.JobTableRight,
                        OutToSlave => "OST_SendRight",
                        xRobotInAuto => "DB_ToHmi".RightRobot.xRobotInAuto,
                        xRobotInManu => "DB_ToHmi".RightRobot.xRobotInManu,
                        xRobotInHome => "DB_ToHmi".xHomePositionR2,
                        xRobotReqReset => "DB_ToHmi".RightRobot.xRobotReqReset,
                        xRobotStopped => "DB_Exchange".xRightRobotStopped,
                        xWarningStart => "DB_Exchange".xStartUpWarningRight,
                        xReqVacuum => "DB_Exchange".xRightRobotStartVacuum,
                        xRecipeInProgress => "DB_ToHmi".RightRobot.xRecipeInProgress,
                        xProductionRunning => "DB_Exchange".xProductionRunningRobot2,
                        xRobotHasStarted => "DB_CommSlave".Right.xRobotHasStarted,
                        xWaitOtherRobotFinished => "DB_CommSlave".Right.xRobotHasFinished,
                        xWaitBothRobotFinished => "DB_CommSlave".Right.xBothSideFinished,
                        xMagazineEmpty => "DB_ToHmi".RightRobot.xMagazineEmpty,
                        xShowPopRemoveDisk => "DB_ToHmi".RightRobot.xShowPopRemoveDisk,
                        xShowPopPickupDisk => "DB_ToHmi".RightRobot.xShowPopPickupDisk,
                        xShowPopFlatnessFault => "DB_ToHmi".RightRobot.xShowPopFlatnessFault,
                        uiJobDataNumber => "DB_ToHmi".RightRobot.uiActualJobDataNumber,
                        xPathInProgress => "DB_ToHmi".RightRobot.xPathInProgress,
                        xPathStopped => "DB_ToHmi".RightRobot.xPathStopped,
                        xPathCancelled => "DB_ToHmi".RightRobot.xPathCancelled,
                        xContactState => "DB_ToHmi".RightRobot.xContactState,
                        xVacValveOpen => "DB_ToHmi".RightRobot.xValveOpen,
                        xVacValveClosed => "DB_ToHmi".RightRobot.xValveClosed,
                        nActualForce => "DB_ToHmi".RightRobot.nActualForce,
                        uiSetSpeed => "DB_ToHmi".RightRobot.uiSetSpeed,
                        uiRobotSpeed => "DB_ToHmi".RightRobot.uiRobotSpeed,
                        uiPaperChangeDistance => "DB_ToHmi".RightRobot.uiPaperChangeDistance,
                        rActualPosition => "DB_ToHmi".RightRobot.rActualPosition,
                        xRangeFinderDetection => "DB_ToHmi".RightRobot.xRangeFinderDetection,
                        uiRangeFinderValue => "DB_ToHmi".RightRobot.uiRangeFinderValue,
                        uiCounterPulse_X => "DB_ToHmi".RightRobot.uiCounterPulse_X,
                        uiCounterPulse_Z => "DB_ToHmi".RightRobot.uiCounterPulse_Z,
                        uiGreaseFault_X => "DB_ToHmi".RightRobot.uiGreaseFault_X,
                        uiGreaseFault_Z => "DB_ToHmi".RightRobot.uiGreaseFault_Z,
                        uiDistanceSandingDisk => "DB_ToHmi".RightRobot.uiDistanceSandingDisk,
                        uiActualRobotSpeed => "DB_ToHmi".RightRobot.uiActualRobotSpeed,
                        udiOdometer_X => "DB_ToHmi".RightRobot.udiOdometer_X,
                        udiOdometer_Z => "DB_ToHmi".RightRobot.udiOdometer_Z,
                        uiDistanceBeforeGreasingX => "DB_ToHmi".RightRobot.uiDistanceBeforeGreasingX,
                        uiDistanceBeforeGreasingZ => "DB_ToHmi".RightRobot.uiDistanceBeforeGreasingZ,
                        uiDiskUsed => "DB_ToHmi".RightRobot.uiNbDiskUsed,
                        uiRobotStatus => "DB_ToHmi".RightRobot.uiRobotStatus,
                        udiFaultTime => "DB_Exchange".RightRobot.udiFaultTime,
                        udiRunTime => "DB_Exchange".RightRobot.udiRunTime,
                        udiPauseTime => "DB_Exchange".RightRobot.udiPauseTime,
                        udiRobotPowerOnTime => "DB_Exchange".RightRobot.udiRobotPowerOnTime,
                        udiRobotDriveOnTime => "DB_Exchange".RightRobot.udiRobotDriveOnTime,
                        bInput100 => "DB_ToHmi".RightRobot.IB_Input100,
                        bInput101 => "DB_ToHmi".RightRobot.IB_Input101,
                        bInput102 => "DB_ToHmi".RightRobot.IB_Input102,
                        bInput103 => "DB_ToHmi".RightRobot.IB_Input103,
                        bInputFast90 => "DB_ToHmi".RightRobot.IB_Fast90,
                        bInputSafety500 => "DB_ToHmi".RightRobot.IB_Safety500,
                        bOutput100 => "DB_ToHmi".RightRobot.OB_Output100,
                        bOutput101 => "DB_ToHmi".RightRobot.OB_Output101,
                        bOutputSafety508 => "DB_ToHmi".RightRobot.OB_Safety508,
                        nInput600 => "DB_ToHmi".RightRobot.IN_Input600,
                        nInput602 => "DB_ToHmi".RightRobot.IN_Input602,
                        nInput604 => "DB_ToHmi".RightRobot.IN_Input604,
                        nInput606 => "DB_ToHmi".RightRobot.IN_Input606,
                        wFaultFerRobotic => "DB_ToHmi".Fault.wFerRoboticRight,
                        wFaultManageRobot => "DB_ToHmi".Fault.wManageRobotRight,
                        wFaultRobot => "DB_ToHmi".Fault.wRobotRight,
                        wFaultOther => "DB_ToHmi".Fault.wOtherRight,
                        wFaultVacuumValve => "DB_ToHmi".Fault.wVacuumValveRight,
                        wFaultFerRoboticManage => "DB_ToHmi".Fault.wFerRoboticManageRight,
                        wWarningDiskTrayEmpty => "DB_ToHmi".Warning.wWarnigRight);
END_REGION

REGION Network 3: Sanding process is in progress
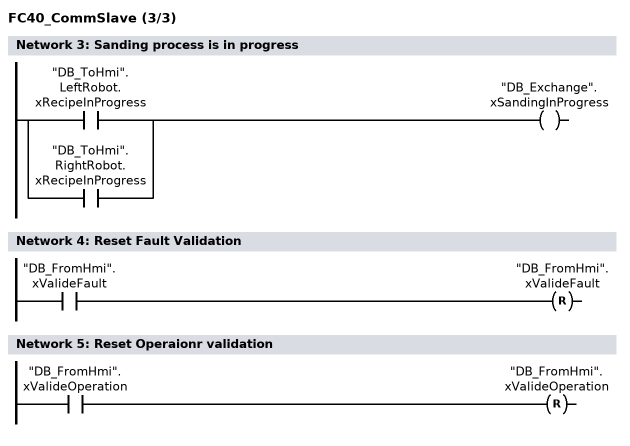
   RUNG wire#powerrail
      Contact( "DB_ToHmi".LeftRobot.xRecipeInProgress )
      wire#w1
      Coil( "DB_Exchange".xSandingInProgress )
   END_RUNG
   RUNG wire#powerrail
      Contact( "DB_ToHmi".RightRobot.xRecipeInProgress )
   END_RUNG wire#w1
   // the same network as SCL:
   "DB_Exchange".xSandingInProgress := "DB_ToHmi".LeftRobot.xRecipeInProgress OR "DB_ToHmi".RightRobot.xRecipeInProgress;
END_REGION

REGION Network 4: Reset Fault Validation
   RUNG wire#powerrail
      Contact( "DB_FromHmi".xValideFault )
      R_Coil( "DB_FromHmi".xValideFault )
   END_RUNG
   // the same network as SCL:
   IF "DB_FromHmi".xValideFault THEN "DB_FromHmi".xValideFault := FALSE; END_IF;
END_REGION

REGION Network 5: Reset Operaionr validation
   RUNG wire#powerrail
      Contact( "DB_FromHmi".xValideOperation )
      R_Coil( "DB_FromHmi".xValideOperation )
   END_RUNG
   // the same network as SCL:
   IF "DB_FromHmi".xValideOperation THEN "DB_FromHmi".xValideOperation := FALSE; END_IF;
END_REGION
END_FUNCTION
